TYPE "EM_Carriage_Brake_State"
VERSION : 0.1
   STRUCT
      state : Int;
      step : Int;
      done : Bool;
      fault : Bool;
   END_STRUCT;
END_TYPE
